(* CODESYS project codesys-dowhile

Project tree, tasks and I/O mapping:
  Device : CODESYS Control Win V3, 3S - Smart Software Solutions GmbH, version 3.5.16.40
    application Application
      libraries: Standard, * (System); VisuDialogs, * (System)
      task MainTask (cyclic, interval t#20ms, priority 1) calls PLC_PRG
      task VISU_TASK (cyclic, interval 100 ms, priority 31) calls VisuElems.Visu_Prg
      program PLC_PRG [ST]
      visualisation Visualization
  text list GlobalTextList
*)

// Device/Application/PLC_PRG
PROGRAM PLC_PRG
VAR
	Start: BOOL:=FALSE;
	Reset: BOOL:=FALSE;
	Timer01: TON;
	Timer02: TON;
	time_out: INT:=10;
END_VAR

WHILE time_out > 0 DO
	Timer01 (IN:= Start AND ( NOT Timer02.Q), PT:=T#300MS);
	Timer02 (IN:= Timer01.Q, PT:=T#500MS);
	IF Timer02.Q THEN
		time_out:= time_out - 1;
	END_IF
	IF Reset THEN
		time_out:=10;
	END_IF
END_WHILE

IF Reset THEN
	time_out:=10;
END_IF

END_PROGRAM

// Device/Application/Visualization
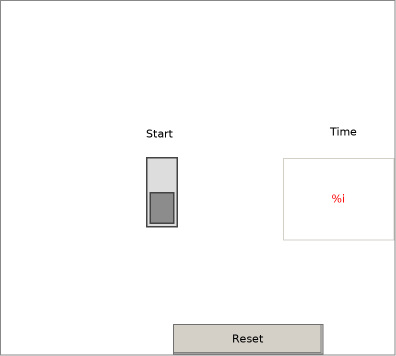
VISUALIZATION Visualization  // 396x356
    DipSwitch (127,157 70x70), variable: PLC_PRG.Start, behaviour: TOGGLE, style: Switch-DipSwitch-Gray
    Label (125,118 69x32), "Start"
    Label (309,116 69x32), "Time"
    Button (173,324 150x30), "Reset"
        tap PLC_PRG.Reset
    Textfield (283,158 111x82), "%i", text variable: PLC_PRG.time_out
END_VISUALIZATION
